{attribute 'qualified_only'}
VAR_GLOBAL
		EtherCAT_Master_ELMxxxx : EtherCAT_Master_ELMxxxx_56F7A9AD;
END_VAR

(* stored: Version 1.2.0.0, ProductVersion 3.1.4024.9
   GVL GVL_iXlinker: Id {61d04bc6-610b-479a-b848-84a07122d871} *)
